TYPE ST_System_BSp_Zustand :
STRUCT
	Betrieb_Anford		: BOOL;
	Betrieb_Soll			: BOOL;
	Betrieb				: BOOL;

	Regelung_Modus		: SINT;
	Regelung_Istw		: REAL;
	Regelung_Sollw		: REAL;

	Modus_Laden				: BOOL;
	Modus_Laden_verfuegbar		: BOOL;
	Modus_Entladen				: BOOL;
	Modus_Entladen_verfuegbar	: BOOL;


	Netze_Anford				: ST_Zustand_Netze_Anford;

	Freigabe				: BOOL;
	Freigabe_Deakt		: BOOL;
	Freigabe_Code		: WORD;

	Stoerung				: BOOL;
	Stoerung_Code		: WORD;

	Warnung				: BOOL;
	Warnung_Code		: WORD;

	Status					: SINT;
	Status_Vorl_Stellventil		: BOOL;
	Status_Vorl_Pumpen		: BOOL;
	Status_Nachl_Stellventil	: BOOL;
	Status_Nachl_Pumpen		: BOOL;
	Status_Wiedereinschalten	: BOOL;
	Temp_oben			: REAL;
	Temp_unten			: REAL;

	Quittierung			: BOOL;

END_STRUCT
END_TYPE

(* stored: Version 1.1.0.1, ProductVersion 3.1.4024.9
   DUT ST_System_BSp_Zustand: Id {24ccefcb-1fee-4a5f-8947-de677ae6d86f} *)
